TYPE Inspection_control :
STRUCT
Buffer_Results_Enable	: BIT ;
Inspection_Results_Ack	: BIT ;
Set_User_Data			: BIT ;
Execute_Command			: BIT ;
Reserved4				: BIT ;
Reserved5				: BIT ;
Reserved6				: BIT ;
Clear_Error				: BIT ;
END_STRUCT
END_TYPE

(* stored: Version 1.1.0.1, ProductVersion 3.1.4024.11
   DUT Inspection_control: Id {ed4c684b-c0bc-414e-b54a-adcd56bdc35c} *)
